# EPICS autosave request: CARSApp/Db/Fluke_8842A_settings.req
# FILE... Fluke_settings.req
$(P)$(M)_Init.AOUT
$(P)$(M)_Read.SCAN
file "scalcout_settings.req", P=$(P)$(M)_Convert
file "scalcout_settings.req", P=$(P)$(M)_Calc
